// TwinCAT 3 PLC project SimpleAlarms
// ProgramVersion: 3.1.4023.0
// libraries:
//   Tc2_Standard, * (Beckhoff Automation GmbH)
//   Tc2_System, * (Beckhoff Automation GmbH)
//   Tc2_Utilities, * (Beckhoff Automation GmbH)
//   Tc3_Module, * (Beckhoff Automation GmbH)
//   VisuDialogs, * (System)
// project tree:
//   DUTs/ ST_EventData.TcDUT
//   / GlobalTextList.TcGTLO, PlcTask.TcTTO, Visualization Manager.TcVMO (not stored), VISU_TASK.TcTTO
//   POUs/ MAIN.TcPOU
//   VISUs/ Event.TcVIS, Visualization.TcVIS
// real-time tasks:
//   TASK PlcTask: cycle T#10ms, priority 20, ADS port 350
//   TASK VISU_TASK: cycle T#200000us, priority 30, ADS port 351

CONFIGURATION SimpleAlarms
    RESOURCE PLC ON TwinCAT3
        TASK PlcTask(INTERVAL := T#10ms, PRIORITY := 20);
        TASK VISU_TASK(INTERVAL := T#200000us, PRIORITY := 30);
        PROGRAM MAIN WITH PlcTask : MAIN;
        PROGRAM VisuElems_Visu_Prg WITH VISU_TASK : VisuElems.Visu_Prg;
    END_RESOURCE
END_CONFIGURATION

// ---- DUTs/ST_EventData.TcDUT
TYPE ST_EventData :
STRUCT
	rVal	:REAL;
	iVal	:INT;;
END_STRUCT
END_TYPE

// ---- POUs/MAIN.TcPOU
PROGRAM MAIN
VAR
	FB_AdsReadEvents_0		: Tc2_Utilities.FB_AdsReadEvents;
	aEvents: ARRAY [1..80] OF Tc2_Utilities.ST_ReadEvent;
	
	Events:ARRAY[1..4]	OF	Tc2_System.FB_SimpleAdsLogEvent;
	temp: REAL;
	ADSLOGEVENT_0: ADSLOGEVENT;
	CfgEvent: TcEvent;
	EventData:ST_EventData;
	TcEventDataFormatString : STRING    := '%f%d';
END_VAR

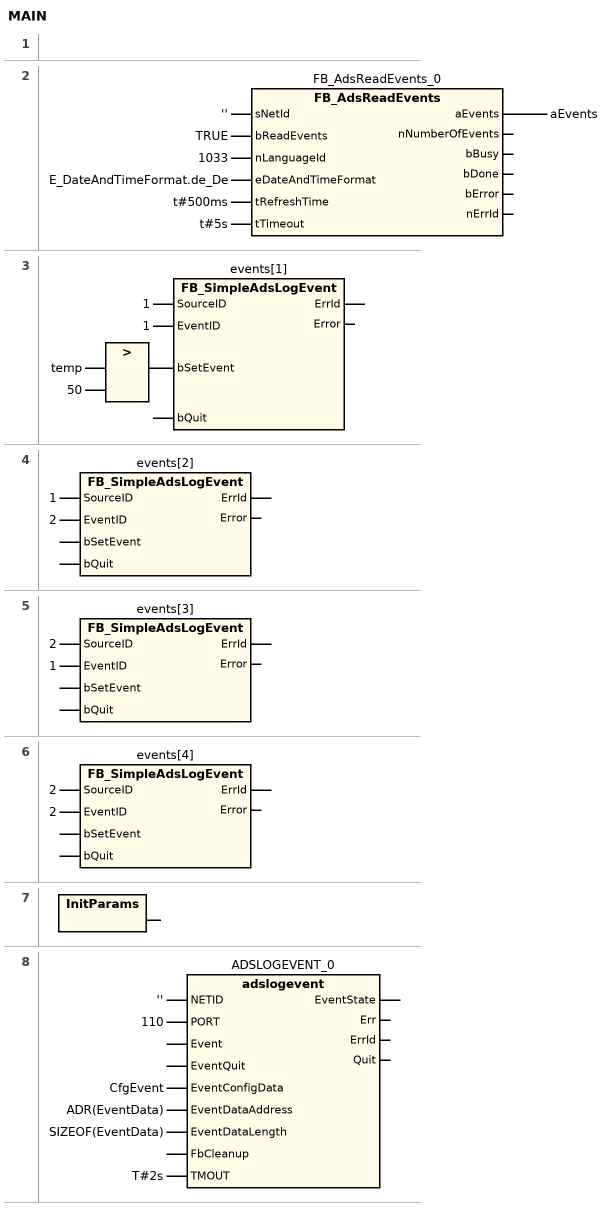
// NETWORK 1

// NETWORK 2
FB_AdsReadEvents_0(
    sNetId := '',
    bReadEvents := TRUE,
    nLanguageId := 1033,
    eDateAndTimeFormat := E_DateAndTimeFormat.de_De,
    tRefreshTime := t#500ms,
    tTimeout := t#5s); // FB_AdsReadEvents
aEvents := FB_AdsReadEvents_0.aEvents;

// NETWORK 3
events[1](SourceID := 1, EventID := 1, bSetEvent := temp > 50); // FB_SimpleAdsLogEvent

// NETWORK 4
events[2](SourceID := 1, EventID := 2); // FB_SimpleAdsLogEvent

// NETWORK 5
events[3](SourceID := 2, EventID := 1); // FB_SimpleAdsLogEvent

// NETWORK 6
events[4](SourceID := 2, EventID := 2); // FB_SimpleAdsLogEvent

// NETWORK 7
InitParams();

// NETWORK 8
ADSLOGEVENT_0(
    NETID := '',
    PORT := 110,
    EventConfigData := CfgEvent,
    EventDataAddress := ADR(EventData),
    EventDataLength := SIZEOF(EventData),
    TMOUT := T#2s); // adslogevent

ACTION InitParams:
//the folowing page explains settings in TcEvent
//https://infosys.beckhoff.com/content/1033/tcplclib_tc2_system/31081227.html?id=6547697951809802698



//CfgEvent.Class := TCEVENTCLASS_ALARM;
//CfgEvent.Prio := 2;
CfgEvent.Id := 1;
CfgEvent.SourceId := 3;
CfgEvent.bQuitRequired := TRUE;
CfgEvent.DataFormatStrAddress := ADR(TcEventDataFormatString);
CfgEvent.Flags := TCEVENTFLAG_LOG OR TCEVENTFLAG_SRCID OR TCEVENTFLAG_AUTOFMTALL;
CfgEvent.StreamType := TCEVENTSTREAM_SIMPLE;
//don't change this 
CfgEvent.ProgId :='TcEventFormatter.TcXMLFormatter' ;



//eventData.rVal     := 2.65;
//eventData.iVal    := 3;
END_ACTION

END_PROGRAM

// ---- GlobalTextList.TcGTLO
TEXTLIST GlobalTextList
  820 = '%d'
  401 = '%d>50?:Event'
  504 = 'aaa'
  464 = 'alarm with parameters'
  710 = 'Error id:%d'
  172 = 'Error id:%x'
  67 = 'Error id:0x%x'
  131 = 'Event %d'
  591 = 'Event 1'
  885 = 'event 1'
  773 = 'Event 2'
  452 = 'event 2'
  834 = 'event2'
  193 = 'Event:Value>50'
  257 = 'Event?:%d>50'
  709 = 'Event?:Value>50'
  642 = 'Evet 1'
  564 = 'Evet i'
  971 = 'float %.2f'
  884 = 'int %i'
  634 = 'quit'
  370 = 'Source %d'
  506 = 'Source 1'
  761 = 'Source 2'
  263 = 'Source 3'
END_TEXTLIST

// ---- VISUs/Event.TcVIS
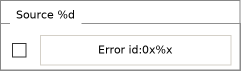
VISUALIZATION Event  // 241x71
VAR_IN_OUT
	Event:FB_SimpleAdsLogEvent;
END_VAR
    GroupBox (0,15 241x56)
        Button (120,20 111x30), "quit"
            tap Event.bQuit
        Textfield (40,20 71x30), "Event %d", text variable: Event.EventID
        Checkbox (10,20 31x30), variable: Event.bSetEvent
        Textfield (40,20 191x30), "Error id:0x%x", text variable: Event.ErrId, colour toggle: Event.Error, invisible if: NOT Event.Error
    Textfield (10,0 71x30), "Source %d", text variable: Event.SourceID
END_VISUALIZATION

// ---- VISUs/Visualization.TcVIS
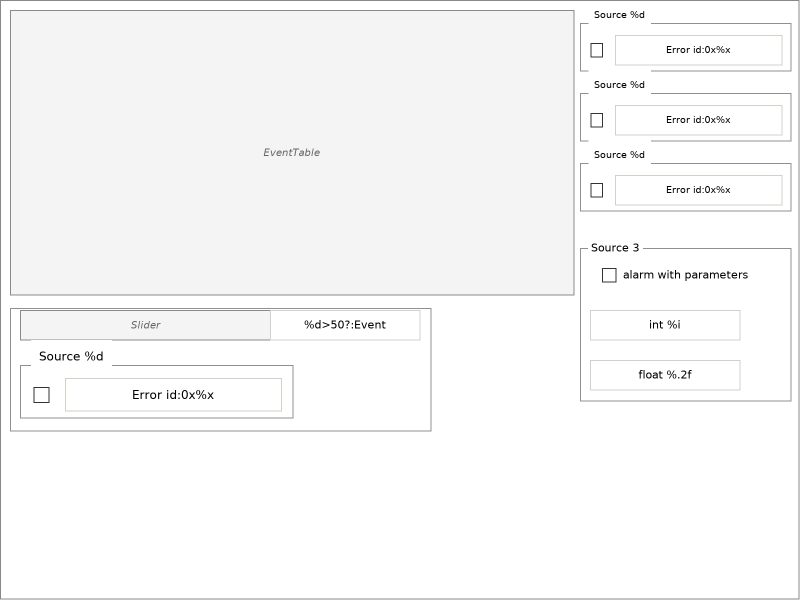
VISUALIZATION Visualization  // 800x600
    EventTable (10,10 564x285)
        p1690906150: Class
        p3258520714: Date
        p2231227367: Time
        p3993844394: Message
        p2076579579: Details
        p3558512729: MAIN.aEvents
        p3921149237: m_pDataArray..pArray
    GroupBox (10,300 421x131)
        Slider (10,10 251x30), variable: MAIN.temp, scale 0..100
        Frame (10,40 273x78)
            shows Event(Event := MAIN.Events[1])
    GroupBox (580,240 211x161), "Source 3"
        Textfield (10,70 150x30), "int %i", text variable: MAIN.EventData.iVal
            OnMouseClick: write the text variable via Default, format %i
        Textfield (10,120 150x30), "float %.2f", text variable: MAIN.EventData.rVal
            OnMouseClick: write the text variable via Default, format %.2f
        Checkbox (20,20 161x30), "alarm with parameters", variable: MAIN.ADSLOGEVENT_0.Event
    Frame (580,0 211x71)
        shows Event(Event := MAIN.Events[2])
    Frame (580,70 211x71)
        shows Event(Event := MAIN.Events[3])
    Frame (580,140 211x71)
        shows Event(Event := MAIN.Events[4])
    Textfield (270,310 150x30), "%d>50?:Event", text variable: MAIN.temp, colour toggle: main.Events[1].bSetEvent
END_VISUALIZATION
